// TIA Portal V17 export
// export: Created 2022-01-04T17:38:19.7883308Z, ExportSetting WithDefaults, DisplayName Totally Integrated Automation Portal, DisplayVersion V17, DisplayName TIA Portal Openness, DisplayVersion V17, DisplayName TIA Portal Version Control Interface, DisplayVersion V17, DisplayName STEP 7 Professional, DisplayVersion V17, DisplayName STEP 7 Safety, DisplayVersion V17, DisplayName WinCC Advanced, DisplayVersion V17
ORGANIZATION_BLOCK "Main"   // OB1, LAD, ProgramCycle
TITLE = "Main Program Sweep (Cycle)"
{ S7_Optimized_Access := 'TRUE' }
VERSION : 0.1
// stored: AutoNumber true, IsIECCheckEnabled false, SetENOAutomatically false
   VAR_INPUT
      Initial_Call : Bool;   // Initial call of this OB
      Remanence : Bool;   // =True, if remanent data are available
   END_VAR
BEGIN

REGION Network 1: Zadanie finałowe kategorii EKSPERT
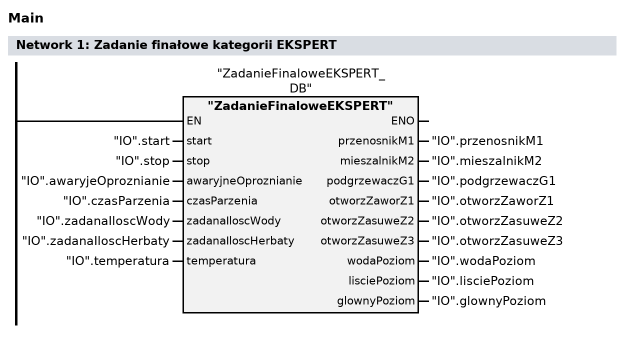
   RUNG wire#powerrail
      "ZadanieFinaloweEKSPERT_DB"(start := "IO".start, stop := "IO".stop, awaryjneOproznianie := "IO".awaryjeOproznianie, czasParzenia := "IO".czasParzenia, zadanaIloscWody := "IO".zadanaIloscWody, zadanaIloscHerbaty := "IO".zadanaIloscHerbaty, temperatura := "IO".temperatura, przenosnikM1 => "IO".przenosnikM1, mieszalnikM2 => "IO".mieszalnikM2, podgrzewaczG1 => "IO".podgrzewaczG1, otworzZaworZ1 => "IO".otworzZaworZ1, otworzZasuweZ2 => "IO".otworzZasuweZ2, otworzZasuweZ3 => "IO".otworzZasuweZ3, wodaPoziom => "IO".wodaPoziom, lisciePoziom => "IO".lisciePoziom, glownyPoziom => "IO".glownyPoziom)
   END_RUNG
   // the same network as SCL:
   "ZadanieFinaloweEKSPERT_DB"(start := "IO".start,   // "ZadanieFinaloweEKSPERT"
                           stop := "IO".stop,
                           awaryjneOproznianie := "IO".awaryjeOproznianie,
                           czasParzenia := "IO".czasParzenia,
                           zadanaIloscWody := "IO".zadanaIloscWody,
                           zadanaIloscHerbaty := "IO".zadanaIloscHerbaty,
                           temperatura := "IO".temperatura,
                           przenosnikM1 => "IO".przenosnikM1,
                           mieszalnikM2 => "IO".mieszalnikM2,
                           podgrzewaczG1 => "IO".podgrzewaczG1,
                           otworzZaworZ1 => "IO".otworzZaworZ1,
                           otworzZasuweZ2 => "IO".otworzZasuweZ2,
                           otworzZasuweZ3 => "IO".otworzZasuweZ3,
                           wodaPoziom => "IO".wodaPoziom,
                           lisciePoziom => "IO".lisciePoziom,
                           glownyPoziom => "IO".glownyPoziom);
END_REGION
END_ORGANIZATION_BLOCK
